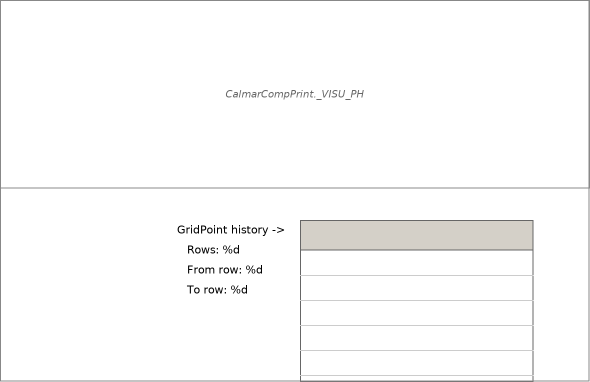
VISUALIZATION _VISU_PH_Grid  // 590x382
VAR_IN_OUT
	m_Inst  : FB_PH_Grid;
END_VAR
    Frame (0,0 590x188)
        shows CalmarCompPrint._VISU_PH(m_Inst := m_Inst)
    Table (300,220 233x162), invisible if: NOT m_Inst.bEnDebug, data array: m_Inst.sPointHistory
        p338671338: m_Inst.sPointHistory[INDEX].dy
        p1892666644: m_Inst.sPointHistory[INDEX].dx
        p3854506369: m_Inst.sPointHistory[INDEX].node
        p1137915858: m_Inst.nPointHead
    Rectangle (174,220 120x20), "GridPoint history ->"
        toggle m_Inst.bEnDebug
    Rectangle (184,240 110x20), "Rows: %d", text variable: m_Inst._nRows, invisible if: NOT m_Inst.bEnDebug
    Rectangle (184,260 110x20), "From row: %d", text variable: m_Inst._nRowLowerBound, invisible if: NOT m_Inst.bEnDebug
    Rectangle (184,280 110x20), "To row: %d", text variable: m_Inst._nRowUpperBound, invisible if: NOT m_Inst.bEnDebug
END_VISUALIZATION

(* stored: Version 1.1.0.1, ProductVersion 3.1.4024.3
   Visu _VISU_PH_Grid: Id {5a227e42-9ee7-45e5-a09a-0bc4696e1119} *)
